FUNCTION_BLOCK PMLStateMachine EXTENDS CyclicBase IMPLEMENTS IPmlStateMachine
VAR_INPUT
END_VAR
VAR_OUTPUT
END_VAR
VAR
	_pmlStateMachine : Tc3_PackML_V2.PML_StateMachine;
	_pmlModeMachine : Tc3_PackML_V2.PML_UnitModeManager;
	_subUnits : ARRAY[0..9] OF IPmlStateMachine;
	subUnitArray : ARRAY[0..9] OF ST_PMLSubUnitInfo;
	_SubUnitReference: ST_PMLSubUnitInfoRef;
	modeChangeTrigger : Tc2_Standard.R_TRIG;
	i: UDINT;
END_VAR

{analysis -2}

METHOD PUBLIC  Cycle : HRESULT
VAR_INPUT
END_VAR
IF _SubUnitReference.NoOfSubUnits <> 0 THEN
	FOR i := 0 TO 9 DO
		IF _subUnits[i] <> 0 THEN
			subUnitArray[i].eState := _subUnits[i].GetCurrentState();
			subUnitArray[i].Active := True;
		END_IF
	END_FOR
	_SubUnitReference.pArray := ADR(subUnitArray);
	_SubUnitReference.ArraySize := SIZEOF(subUnitArray);
END_IF

_pmlStateMachine(eMode := _pmlModeMachine.eModeStatus, stSubUnitInfoRef := _SubUnitReference);
_pmlModeMachine(eState := _pmlStateMachine.eState, bExecute := modeChangeTrigger.Q);
modeChangeTrigger();
Cycle := S_OK;
END_METHOD

METHOD PUBLIC GetCurrentMode : E_PmlProtectedUnitMode
VAR_INPUT
END_VAR
GetCurrentMode := _pmlModeMachine.eModeStatus;
END_METHOD

METHOD PUBLIC GetCurrentState : E_PMLState
VAR_INPUT
END_VAR
GetCurrentState := _pmlStateMachine.eState;
END_METHOD

METHOD PUBLIC PmlModeCommand : Bool
VAR_INPUT
	Mode : E_PMLProtectedUnitMode;
END_VAR
_pmlModeMachine.eModeCommand := Mode;
modeChangeTrigger.CLK := TRUE;
PmlModeCommand := TRUE;
END_METHOD

METHOD PUBLIC PmlStateCommand : BOOL
VAR_INPUT
	Command : E_PMLCommand;
END_VAR
_pmlStateMachine.eCommand := Command;
PmlStateCommand := TRUE;
END_METHOD

METHOD PUBLIC RegisterSubUnit : IPmlStateMachine
VAR_INPUT
	SubUnit : IPmlStateMachine;
END_VAR
FOR i := 0 TO 9 DO
	IF _subUnits[i] = 0 THEN
		_subUnits[i] := SubUnit;
		_SubUnitReference.NoOfSubUnits := i + 1;
		EXIT;
	END_IF
END_FOR
END_METHOD

METHOD PUBLIC SetStateComplete : BOOL
VAR_INPUT
END_VAR
_pmlStateMachine.M_StateComplete();
SetStateComplete := TRUE;
END_METHOD

END_FUNCTION_BLOCK

(* stored: Version 1.1.0.1
   POU PMLStateMachine: Id {516e0c08-a37e-42cd-8e77-8f251b5a3702}, SpecialFunc None
   Method Cycle: Id {bacdfbc6-974d-4c0e-ad97-1906ab402beb}
   Method GetCurrentMode: Id {f7905c4c-714b-498b-b04c-920a1380f7b9}
   Method GetCurrentState: Id {937de08d-f59f-4669-8328-29a92bad08ed}
   Method PmlModeCommand: Id {7d221af2-3765-4e6f-948f-c319a462fce9}
   Method PmlStateCommand: Id {e72652e0-73b2-4e23-9575-4c2cc8e1653b}
   Method RegisterSubUnit: Id {e84e1125-c3e0-45d6-bfd5-89e06f8482f4}
   Method SetStateComplete: Id {65676236-1b0c-487c-a08c-78c21658a2d0} *)
